// Mitsubishi GX Works2 project: 230927-007-A1+A2.A3   PLC: Q03UDV

// task Task_01 (event TRUE, interval 0, priority 31): POU_01

PROGRAM POU_01
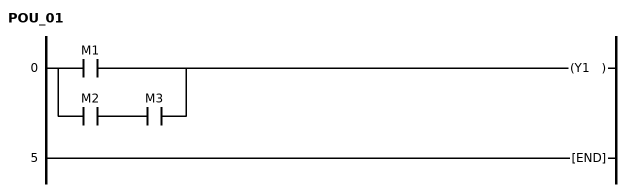
0     LD      M1
      LD      M2
      AND     M3
      ORB
      OUT     Y1
5     END
END_PROGRAM
